TYPE ST_MESSAGE_CTRL :
STRUCT
  Cmd         : E_MESSAGE_CTRL;
END_STRUCT
END_TYPE

(* stored: Version 1.1.0.1
   DUT ST_MESSAGE_CTRL: Id {0f3b2dcd-3897-4405-b1e4-0ff57326ad99} *)
